FUNCTION_BLOCK TcoSequenceAutoRestorableTest EXTENDS TcoCore._internals_TcoContext
VAR
	_callMyPlcInstance	:	BOOL := FALSE;
	_sequencer : _TcoSequence(THIS^, eRestoreMode.AutoRestoreMembers);
	_runPLCinstanceOnce : BOOL := FALSE;
	_runPLCinstanceCyclicaly : BOOL := FALSE;
	_stepID : INT := 32764;
	_enabled : BOOL;
	_stepDescription : STRING := 'Last step sequence message';	
	_runOneStep : BOOL;
	_runAllSteps : BOOL;
	_finishStep : BOOL;
	_restore : BOOL;
	_cycleCount : INT;
	_restoreCycleCount : INT;
	_init: BOOL;
	_setCurrentStepPropTestData : TcoCore.StepDetails;
END_VAR

IF _callMyPlcInstance THEN
	IF NOT _init THEN
		ContextOpen();	
		ContextClose();	
		_init := THIS^._rtc.IsValid;
	END_IF
	
	IF _restore THEN
		ContextOpen();	
		THIS^._sequencer.Restore();	
		_restoreCycleCount := _restoreCycleCount + 1;
		_restore := FALSE;
		ContextClose();	
		RETURN;
	END_IF
	
	IF _runPLCinstanceOnce AND NOT _runPLCinstanceCyclicaly THEN
		ContextOpen();	
		THIS^.PLCinstanceRun(_stepID , _enabled, _stepDescription);
		_cycleCount := _cycleCount + 1;
		_runPLCinstanceOnce := FALSE;
		ContextClose();	
	END_IF
	
	IF _runPLCinstanceCyclicaly AND NOT _runPLCinstanceOnce THEN
		ContextOpen();	
		THIS^.PLCinstanceRun(_stepID , _enabled, _stepDescription);
		_cycleCount := _cycleCount + 1;
		ContextClose();	
	END_IF
END_IF;

{attribute 'TcRpcEnable'}
METHOD ChildHasAutoRestoreEnabled : BOOL;
ChildHasAutoRestoreEnabled := _sequencer.ChildHasAutoRestoreEnabled();
END_METHOD

{attribute 'TcRpcEnable'}
METHOD ChildIsAutoRestorable : BOOL;
ChildIsAutoRestorable := _sequencer.ChildIsAutoRestorable();
END_METHOD

{attribute 'TcRpcEnable'}
METHOD CleanupPointers
_sequencer.CleanupPointers();
END_METHOD

{attribute 'TcRpcEnable'}
METHOD ClearNumberOfSteps
_sequencer.ClearNumberOfSteps();
END_METHOD

{attribute 'TcRpcEnable'}
METHOD PROTECTED ContextClose
SUPER^._Close();
END_METHOD

{attribute 'TcRpcEnable'}
METHOD ContextOpen
SUPER^._Open();
END_METHOD

{attribute 'TcRpcEnable'}
METHOD GetChildState : INT
GetChildState := _sequencer.GetChildState();
END_METHOD

{attribute 'TcRpcEnable'}
METHOD GetCurrentStepOrder : UINT
GetCurrentStepOrder := _sequencer._currentStep.Order;
END_METHOD

{attribute 'TcRpcEnable'}
METHOD GetCurrentStepPropTest
_setCurrentStepPropTestData := THIS^._sequencer.CurrentStep;
END_METHOD

{attribute 'TcRpcEnable'}
METHOD GetNumberOfStepsInSequence : UINT
GetNumberOfStepsInSequence := _sequencer._numberOfStepsInSequence;
END_METHOD

{attribute 'TcRpcEnable'}
METHOD GetOrderOfTheCurrentlyEvaluatedStep : UINT
GetOrderOfTheCurrentlyEvaluatedStep := _sequencer._theOrderOfTheCurrentlyEvaluatedStep;
END_METHOD

{attribute 'TcRpcEnable'}
METHOD GetOrderOfTheCurrentlyExecutedStep : UINT
GetOrderOfTheCurrentlyExecutedStep := _sequencer._theOrderOfTheCurrentlyExecutedStep;
END_METHOD

{attribute 'TcRpcEnable'}
METHOD GetPreviousNumberOfStepsInSequence : UINT
GetPreviousNumberOfStepsInSequence := _sequencer._previousNumberOfStepsInSequence;
END_METHOD

{attribute 'TcRpcEnable'}
METHOD GetRequestStepCycle : UINT
GetRequestStepCycle := _sequencer.RequestStepCycle;
END_METHOD

{attribute 'TcRpcEnable'}
METHOD GetSequencerErrorId : INT
GetSequencerErrorId := _sequencer.GetSequencerErrorId();
END_METHOD

{attribute 'TcRpcEnable'}
METHOD GetTextOfTheMostImportantMessage : STRING(254)
GetTextOfTheMostImportantMessage := THIS^._sequencer.GetTextOfTheMostImportantMessage();
END_METHOD

{attribute 'TcRpcEnable'}
METHOD HasAutoRestoreEnabled : BOOL;
HasAutoRestoreEnabled := _sequencer.HasAutoRestoreEnabled();
END_METHOD

{attribute 'TcRpcEnable'}
METHOD IsAutoRestorable : BOOL;
IsAutoRestorable := _sequencer.IsAutoRestorable();
END_METHOD

{attribute 'TcRpcEnable'}
METHOD IsFirstStepEntry : BOOL
IsFirstStepEntry := THIS^._sequencer.IsFirstStepEntry();
END_METHOD

METHOD PROTECTED  Main
END_METHOD

{attribute 'TcRpcEnable'}
METHOD PLCinstanceRun
VAR_INPUT
	inStepId			:	UINT;
	inEnabled			:	BOOL;
	inStepDescription	:	STRING(254);	
END_VAR
THIS^._sequencer.SetTestParams(	_runOneStep , _runAllSteps , _finishStep , inStepId , inEnabled , inStepDescription);

THIS^._sequencer._RunExecutionSubstitute();
END_METHOD

{attribute 'TcRpcEnable'}
METHOD RequestStep
VAR_INPUT
	inRequestedStepId : INT;
END_VAR
_sequencer._RequestStep(inRequestedStepId);
END_METHOD

{attribute 'TcRpcEnable'}
METHOD Restore
_sequencer.Restore();
END_METHOD

{attribute 'TcRpcEnable'}
METHOD SequenceComplete
_sequencer._SequenceComplete();
END_METHOD

{attribute 'TcRpcEnable'}
METHOD SequencerClose
THIS^._sequencer.SequencerClose();
END_METHOD

{attribute 'TcRpcEnable'}
METHOD SequencerHasError : BOOL
SequencerHasError := _sequencer.SequencerHasError();
END_METHOD

{attribute 'TcRpcEnable'}
METHOD SequencerOpen
THIS^._sequencer.SequencerOpen();
END_METHOD

{attribute 'TcRpcEnable'}
METHOD SetChildState
VAR_INPUT
	inState			:	INT;
END_VAR
_sequencer.SetChildState(inState);
END_METHOD

{attribute 'TcRpcEnable'}
METHOD SetCurrentStep
VAR_INPUT
	inStepID 			:	INT;
	inStepDescription	:	STRING(254);
END_VAR
_sequencer.SetCurrentStep(inStepID := inStepID, inStepDescription := inStepDescription);
END_METHOD

{attribute 'TcRpcEnable'}
METHOD SetCurrentStepToErrorState : BOOL
SetCurrentStepToErrorState := _sequencer.SetCurrentStepToErrorState();
END_METHOD

{attribute 'TcRpcEnable'}
METHOD SetCyclicMode : BOOL
SetCyclicMode := _sequencer.SetCyclicMode();
END_METHOD

{attribute 'TcRpcEnable'}
METHOD SetInvalidMode : BOOL
SetInvalidMode := _sequencer.SetInvalidMode();
END_METHOD

{attribute 'TcRpcEnable'}
METHOD SetNumberOfSteps : UINT
VAR_INPUT
	inNumberOfSteps :UINT;
END_VAR
_sequencer.SetNumberOfSteps(inNumberOfSteps);
SetNumberOfSteps := _sequencer._numberOfStepsInSequence;
END_METHOD

{attribute 'TcRpcEnable'}
METHOD SetRequestStepCycle : UINT
VAR_INPUT
	Value : UINT;
END_VAR
_sequencer.RequestStepCycle := Value;

SetRequestStepCycle := _sequencer.RequestStepCycle;
END_METHOD

{attribute 'TcRpcEnable'}
METHOD SetSequenceAsChecked : BOOL
VAR_INPUT
END_VAR
_sequencer.SetSequenceAsChecked();
END_METHOD

{attribute 'TcRpcEnable'}
METHOD SetSequenceAsNotChecked : BOOL
VAR_INPUT
END_VAR
_sequencer.SetSequenceAsNotChecked();
END_METHOD

{attribute 'TcRpcEnable'}
METHOD SetStepMode : BOOL
SetStepMode := _sequencer.SetStepMode();
END_METHOD

{attribute 'TcRpcEnable'}
METHOD Step : BOOL
VAR_INPUT
	inStepId			:	INT;
	inEnabled			:	BOOL;
	inStepDescription	:	STRING(254);		
END_VAR
Step := _sequencer._Step(inStepID := inStepId, inEnabled := inEnabled, inStepDescription := inStepDescription);
END_METHOD

{attribute 'TcRpcEnable'}
METHOD StepBackward
_sequencer._StepBackward();
END_METHOD

{attribute 'TcRpcEnable'}
METHOD StepCompleteWhen 
VAR_INPUT
	inCondition : BOOL;
END_VAR
_sequencer._StepCompleteWhen(inCondition);
END_METHOD

{attribute 'TcRpcEnable'}
METHOD StepForward
_sequencer._StepForward();
END_METHOD

{attribute 'TcRpcEnable'}
METHOD StepIn
_sequencer._StepIn();
END_METHOD

{attribute 'TcRpcEnable'}
METHOD UpdateCurrentStepDetails
VAR_INPUT
END_VAR
_sequencer.UpdateCurrentStepDetails();
END_METHOD

END_FUNCTION_BLOCK

(* stored: Version 1.1.0.1
   POU TcoSequenceAutoRestorableTest: Id {da1e6e89-a289-01aa-206d-d93ce5f0512f}, SpecialFunc None
   Method ChildHasAutoRestoreEnabled: Id {09469517-459e-0a54-3500-4f68e2b134f9}
   Method ChildIsAutoRestorable: Id {59881bf6-c411-0622-30ce-413c64f3623c}
   Method CleanupPointers: Id {19a29486-60c8-0c17-09bc-f75411157235}
   Method ClearNumberOfSteps: Id {84b41c04-39dc-00ea-34ed-b569a001f6d5}
   Method ContextClose: Id {c69371ab-2b05-0fd2-37d6-b5b2127462be}
   Method ContextOpen: Id {817ef04d-0b08-0f01-0ded-bb2d74814989}
   Method GetChildState: Id {a9d53ecc-bb74-0d1c-29a8-98c406a651cf}
   Method GetCurrentStepOrder: Id {bf6c0671-c89e-0807-02ea-3dfbfa2c7dfc}
   Method GetCurrentStepPropTest: Id {ede823ca-ab35-08ad-2372-794e1981362f}
   Method GetNumberOfStepsInSequence: Id {e60e7296-6db8-00c9-0b69-45e219b52b28}
   Method GetOrderOfTheCurrentlyEvaluatedStep: Id {0d1e8fea-daab-08c5-2878-ac2770aa9bb2}
   Method GetOrderOfTheCurrentlyExecutedStep: Id {8ff01e8e-d785-0c66-1af7-8c85b277a841}
   Method GetPreviousNumberOfStepsInSequence: Id {95f835a2-ac62-0d14-2d18-25fd9bc36c86}
   Method GetRequestStepCycle: Id {2440d551-76f9-00a9-366a-168689cd3f30}
   Method GetSequencerErrorId: Id {f348bc9d-b9e6-0266-190e-287675a7866c}
   Method GetTextOfTheMostImportantMessage: Id {7ae1dca5-b867-0b6a-17f7-1b54f628395e}
   Method HasAutoRestoreEnabled: Id {bcf3f5a8-6e78-032b-219e-d7072589ba60}
   Method IsAutoRestorable: Id {8912a703-8973-01a1-1be3-0597339c58bc}
   Method IsFirstStepEntry: Id {c9a17177-2f8e-0af0-2b90-d89012645be6}
   Method Main: Id {781f0596-be3d-0794-1f89-6ab5bcb19c7d}
   Method PLCinstanceRun: Id {17b14b57-b647-0ed4-01c8-7bd03d5382c3}
   Method RequestStep: Id {6d0ec76f-4ba0-08c9-01cd-cea37080166c}
   Method Restore: Id {65dc9fc3-4844-0c49-19d4-5ee8c4258091}
   Method SequenceComplete: Id {d4e2486d-f3a6-03cb-3df8-571d1b8eb133}
   Method SequencerClose: Id {78cd2ee0-9f1b-029a-1354-ff3f09ef71c1}
   Method SequencerHasError: Id {d7ab3537-f6a7-0bc7-33aa-2cb955b12d30}
   Method SequencerOpen: Id {24c115dd-0724-0cbb-107b-46ace34760ed}
   Method SetChildState: Id {71c3d726-df7b-0651-21fd-5b3aa047ec91}
   Method SetCurrentStep: Id {3a4cf92b-1bd2-0808-35c6-78b4da513418}
   Method SetCurrentStepToErrorState: Id {132d2f99-20d3-0d03-0a4e-5b512182b0f5}
   Method SetCyclicMode: Id {b5acae6e-eb14-022f-3bb5-cc54e2210820}
   Method SetInvalidMode: Id {41814ef8-dcc6-006d-27c3-14989b56cc8e}
   Method SetNumberOfSteps: Id {25bafa5e-ecbf-02be-37c9-f079d9ee1692}
   Method SetRequestStepCycle: Id {9a79e7f9-7132-0438-2455-c72bc25502e9}
   Method SetSequenceAsChecked: Id {0d202217-8329-0b24-25cd-e4be9ed0e7da}
   Method SetSequenceAsNotChecked: Id {e47e466c-ef7c-0596-2d1b-23eb85577608}
   Method SetStepMode: Id {71dd69b4-0c2f-09e2-26dc-070dab20e5e7}
   Method Step: Id {2c196d81-8e5b-03dc-31bf-3eb26c1a2ad6}
   Method StepBackward: Id {31d10c76-36d0-0ada-02c9-31d4274a0faf}
   Method StepCompleteWhen: Id {d2e36709-8bee-0409-3fd5-61a221ad1f14}
   Method StepForward: Id {e07068ea-68d5-0aed-25d4-4639a290a714}
   Method StepIn: Id {8b6aa015-5969-0851-2c25-e56f408a3db8}
   Method UpdateCurrentStepDetails: Id {9f07f641-bdc9-0a95-0492-e082e9ec9e4f} *)
